FUNCTION F_SAFETY_StatusFB_TO_OPMODE : ST_SAFETY_FBOPMODE
VAR_INPUT
	stFBStatus						: ST_SAFETY_FBStatus; 	(* Struktura ogolna *)
END_VAR

F_SAFETY_StatusFB_TO_OPMODE.uStatus.stStatusWords	:= stFBStatus;									(* Przepisanie *)
F_SAFETY_StatusFB_TO_OPMODE.eState 					:= stFBStatus.BState;							(* Ustawienie enum *)
F_SAFETY_StatusFB_TO_OPMODE.bGeneralError			:= stFBStatus.wDiagnosis <> 0;					(* General Error *)

END_FUNCTION

(* stored: Version 1.1.0.1, ProductVersion 3.1.4022.12
   POU F_SAFETY_StatusFB_TO_OPMODE: Id {b56a960b-cfd1-45e5-8235-b04b300e6766}, SpecialFunc None *)
